// LS Electric XG5000 project: LoadWizardPro_v2
// PLC LoadWizardPLC
// module base 0 slot 0: FEnet:XGL-EFMT(B) (Fast Ethernet Module, Electrical Master)
// module base 0 slot 1: Input Module:XGI-D22A/B (DC 24V Input, 16 Contacts)
// module base 0 slot 2: Output Module:XGQ-TR2A/B (Transistor Output, 16 Contacts (0.5A, Sink Output/Source Output))
// module base 0 slot 3: Input Module:XGI-D22A/B (DC 24V Input, 16 Contacts)
// module base 0 slot 4: Output Module:XGQ-RY2A/B (Relay Output, 16 Contacts (2A, No Varistor/Varistor))

PROGRAM Main (task: Scan Program)

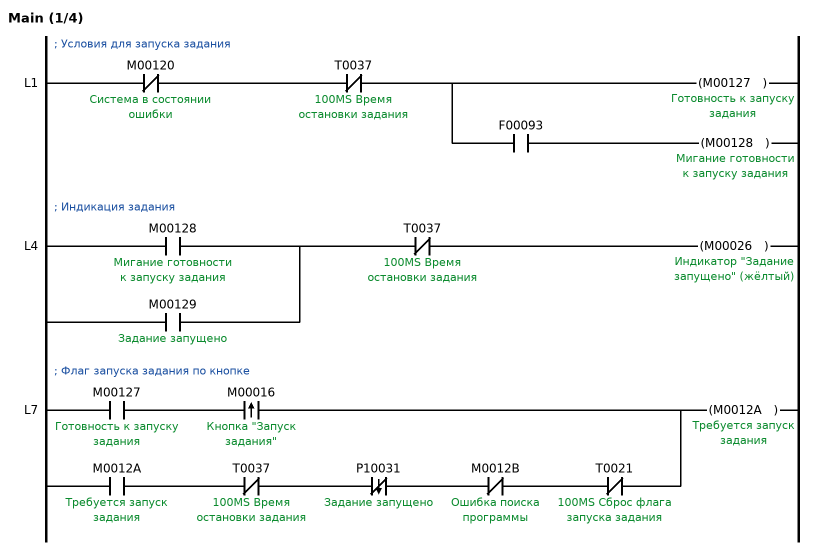
// Условия для запуска задания
; L1
LOAD NOT  M00120	// Система в состоянии ошибки
AND NOT   T0037	// 100MS Время остановки задания
OUT       M00127	// Готовность к запуску задания
AND       F00093
OUT       M00128	// Мигание готовности к запуску задания
// Индикация задания
; L4
LOAD      M00128	// Мигание готовности к запуску задания
OR        M00129	// Задание запущено
AND NOT   T0037	// 100MS Время остановки задания
OUT       M00026	// Индикатор "Задание запущено" (жёлтый)
// Флаг запуска задания по кнопке
; L7
LOAD      M00127	// Готовность к запуску задания
ANDP      M00016	// Кнопка "Запуск задания"
LOAD      M0012A	// Требуется запуск задания
AND NOT   T0037	// 100MS Время остановки задания
ANDN NOT  P10031	// Задание запущено
AND NOT   M0012B	// Ошибка поиска программы
AND NOT   T0021	// 100MS Сброс флага запуска задания
OR LOAD
OUT       M0012A	// Требуется запуск задания

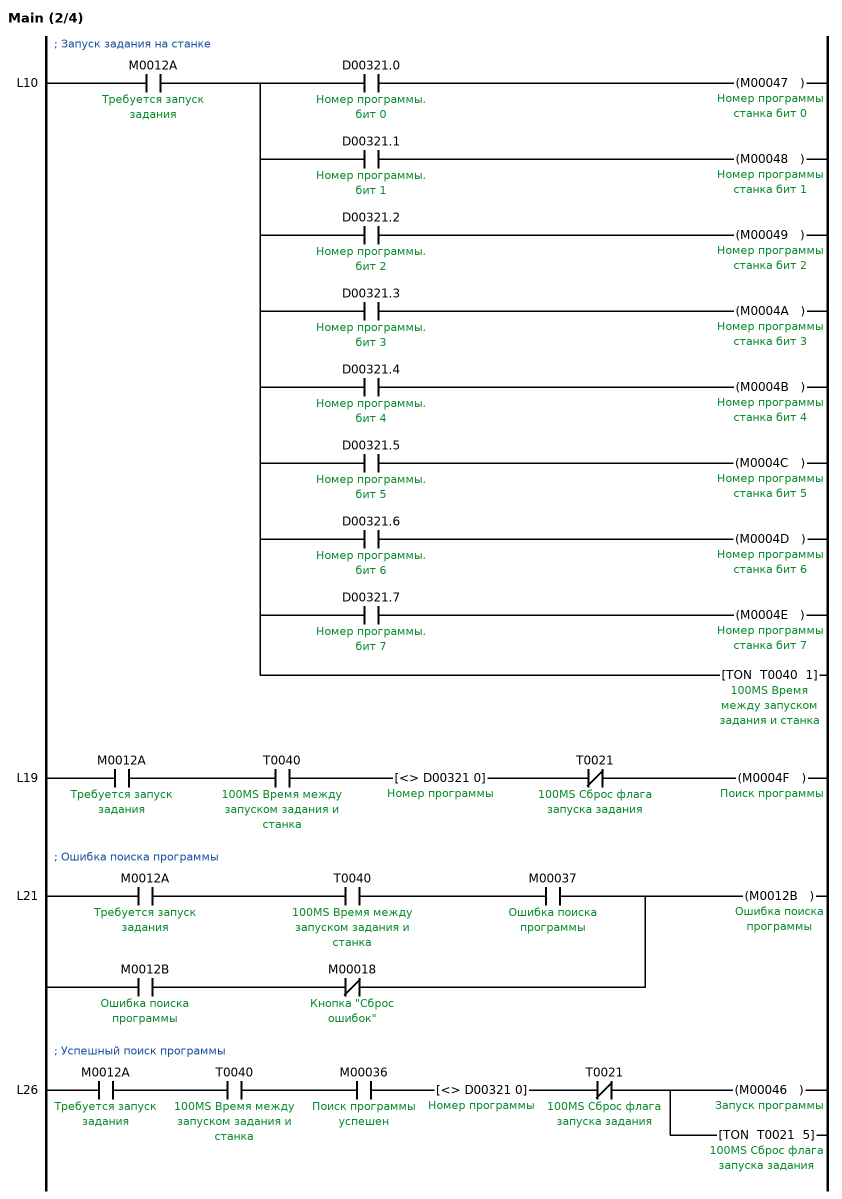
// Запуск задания на станке
; L10
LOAD      M0012A	// Требуется запуск задания
MPUSH
AND       D00321.0	// Номер программы. бит 0
OUT       M00047	// Номер программы станка бит 0
MLOAD
AND       D00321.1	// Номер программы. бит 1
OUT       M00048	// Номер программы станка бит 1
MLOAD
AND       D00321.2	// Номер программы. бит 2
OUT       M00049	// Номер программы станка бит 2
MLOAD
AND       D00321.3	// Номер программы. бит 3
OUT       M0004A	// Номер программы станка бит 3
MLOAD
AND       D00321.4	// Номер программы. бит 4
OUT       M0004B	// Номер программы станка бит 4
MLOAD
AND       D00321.5	// Номер программы. бит 5
OUT       M0004C	// Номер программы станка бит 5
MLOAD
AND       D00321.6	// Номер программы. бит 6
OUT       M0004D	// Номер программы станка бит 6
MLOAD
AND       D00321.7	// Номер программы. бит 7
OUT       M0004E	// Номер программы станка бит 7
MPOP
TON       T0040 1	// 100MS Время между запуском задания и станка
; L19
LOAD      M0012A	// Требуется запуск задания
AND       T0040	// 100MS Время между запуском задания и станка
AND<>     D00321 0	// Номер программы
AND NOT   T0021	// 100MS Сброс флага запуска задания
OUT       M0004F	// Поиск программы
// Ошибка поиска программы
; L21
LOAD      M0012A	// Требуется запуск задания
AND       T0040	// 100MS Время между запуском задания и станка
AND       M00037	// Ошибка поиска программы
LOAD      M0012B	// Ошибка поиска программы
AND NOT   M00018	// Кнопка "Сброс ошибок"
OR LOAD
OUT       M0012B	// Ошибка поиска программы
// Успешный поиск программы
; L26
LOAD      M0012A	// Требуется запуск задания
AND       T0040	// 100MS Время между запуском задания и станка
AND       M00036	// Поиск программы успешен
AND<>     D00321 0	// Номер программы
AND NOT   T0021	// 100MS Сброс флага запуска задания
OUT       M00046	// Запуск программы
TON       T0021 5	// 100MS Сброс флага запуска задания

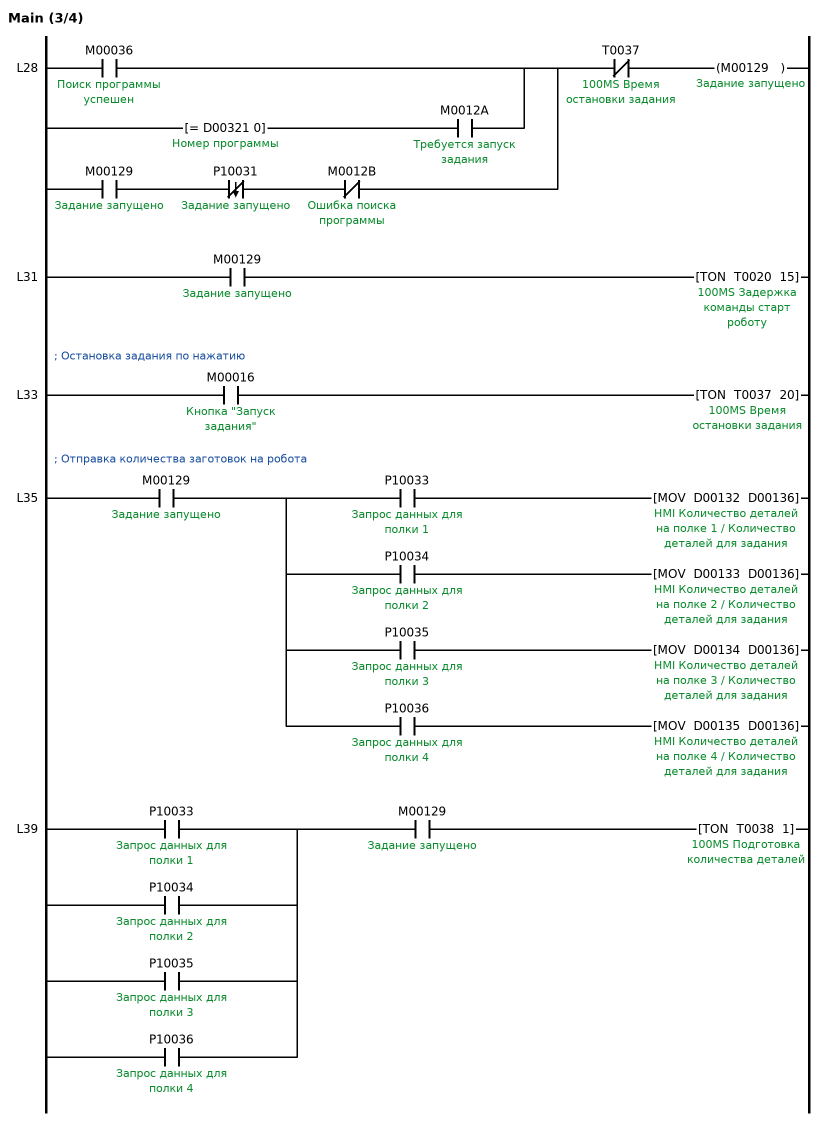
; L28
LOAD      M00036	// Поиск программы успешен
LOAD=     D00321 0	// Номер программы
AND       M0012A	// Требуется запуск задания
OR LOAD
LOAD      M00129	// Задание запущено
ANDN NOT  P10031	// Задание запущено
AND NOT   M0012B	// Ошибка поиска программы
OR LOAD
AND NOT   T0037	// 100MS Время остановки задания
OUT       M00129	// Задание запущено
; L31
LOAD      M00129	// Задание запущено
TON       T0020 15	// 100MS Задержка команды старт роботу
// Остановка задания по нажатию
; L33
LOAD      M00016	// Кнопка "Запуск задания"
TON       T0037 20	// 100MS Время остановки задания
// Отправка количества заготовок на робота
; L35
LOAD      M00129	// Задание запущено
MPUSH
AND       P10033	// Запрос данных для полки 1
MOV       D00132 D00136	// HMI Количество деталей на полке 1 / Количество деталей для задания
MLOAD
AND       P10034	// Запрос данных для полки 2
MOV       D00133 D00136	// HMI Количество деталей на полке 2 / Количество деталей для задания
MLOAD
AND       P10035	// Запрос данных для полки 3
MOV       D00134 D00136	// HMI Количество деталей на полке 3 / Количество деталей для задания
MPOP
AND       P10036	// Запрос данных для полки 4
MOV       D00135 D00136	// HMI Количество деталей на полке 4 / Количество деталей для задания
; L39
LOAD      P10033	// Запрос данных для полки 1
OR        P10034	// Запрос данных для полки 2
OR        P10035	// Запрос данных для полки 3
OR        P10036	// Запрос данных для полки 4
AND       M00129	// Задание запущено
TON       T0038 1	// 100MS Подготовка количества деталей

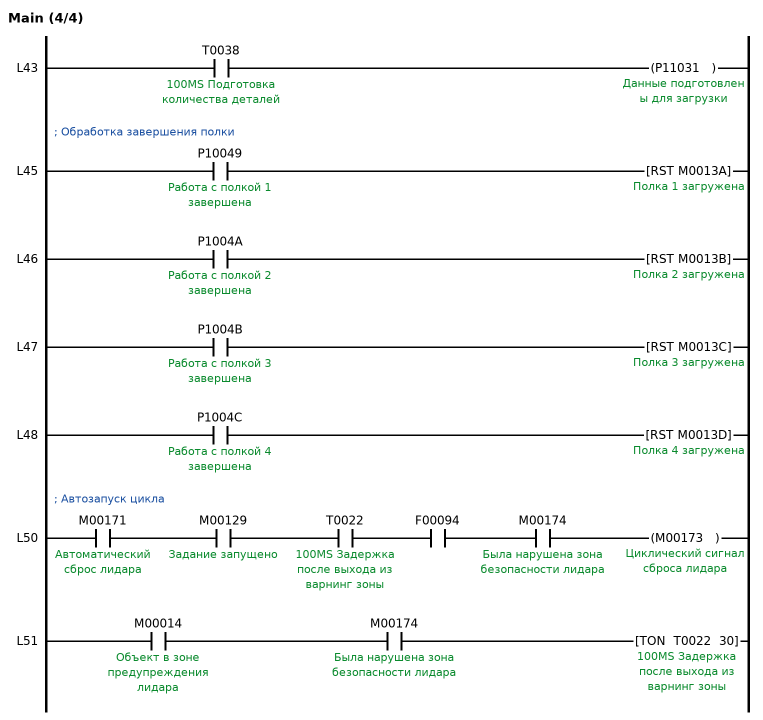
; L43
LOAD      T0038	// 100MS Подготовка количества деталей
OUT       P11031	// Данные подготовлены для загрузки
// Обработка завершения полки
; L45
LOAD      P10049	// Работа с полкой 1 завершена
RST       M0013A	// Полка 1 загружена
; L46
LOAD      P1004A	// Работа с полкой 2 завершена
RST       M0013B	// Полка 2 загружена
; L47
LOAD      P1004B	// Работа с полкой 3 завершена
RST       M0013C	// Полка 3 загружена
; L48
LOAD      P1004C	// Работа с полкой 4 завершена
RST       M0013D	// Полка 4 загружена
// Автозапуск цикла
; L50
LOAD      M00171	// Автоматический сброс лидара
AND       M00129	// Задание запущено
AND       T0022	// 100MS Задержка после выхода из варнинг зоны
AND       F00094
AND       M00174	// Была нарушена зона безопасности лидара
OUT       M00173	// Циклический сигнал сброса лидара
; L51
LOAD      M00014	// Объект в зоне предупреждения лидара
AND       M00174	// Была нарушена зона безопасности лидара
TON       T0022 30	// 100MS Задержка после выхода из варнинг зоны

PROGRAM Robot (task: Scan Program)

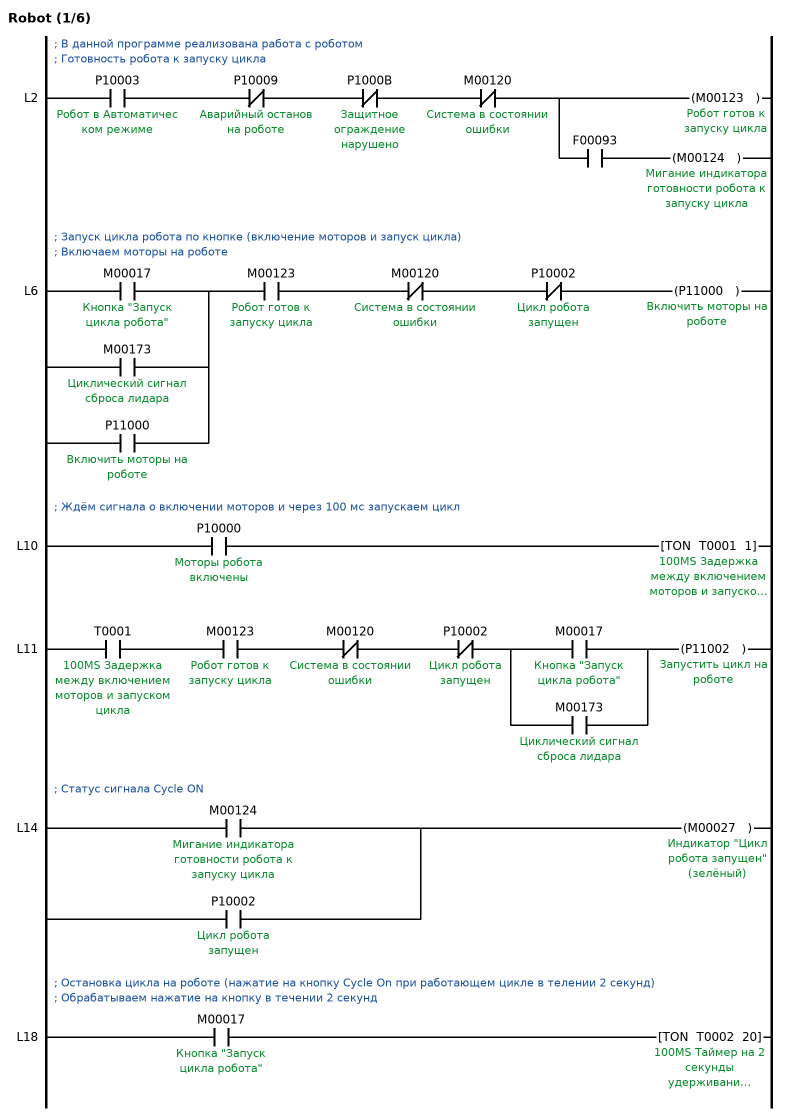
// В данной программе реализована работа с роботом
// Готовность робота к запуску цикла
; L2
LOAD      P10003	// Робот в Автоматическом режиме
AND NOT   P10009	// Аварийный останов на роботе
AND NOT   P1000B	// Защитное ограждение нарушено
AND NOT   M00120	// Система в состоянии ошибки
OUT       M00123	// Робот готов к запуску цикла
AND       F00093
OUT       M00124	// Мигание индикатора готовности робота к запуску цикла
// Запуск цикла робота по кнопке (включение моторов и запуск цикла)
// Включаем моторы на роботе
; L6
LOAD      M00017	// Кнопка "Запуск цикла робота"
OR        M00173	// Циклический сигнал сброса лидара
OR        P11000	// Включить моторы на роботе
AND       M00123	// Робот готов к запуску цикла
AND NOT   M00120	// Система в состоянии ошибки
AND NOT   P10002	// Цикл робота запущен
OUT       P11000	// Включить моторы на роботе
// Ждём сигнала о включении моторов и через 100 мс запускаем цикл
; L10
LOAD      P10000	// Моторы робота включены
TON       T0001 1	// 100MS Задержка между включением моторов и запуском цикла
; L11
LOAD      T0001	// 100MS Задержка между включением моторов и запуском цикла
AND       M00123	// Робот готов к запуску цикла
AND NOT   M00120	// Система в состоянии ошибки
AND NOT   P10002	// Цикл робота запущен
LOAD      M00017	// Кнопка "Запуск цикла робота"
OR        M00173	// Циклический сигнал сброса лидара
AND LOAD
OUT       P11002	// Запустить цикл на роботе
// output comment: 
// Статус сигнала Cycle ON
; L14
LOAD      M00124	// Мигание индикатора готовности робота к запуску цикла
OR        P10002	// Цикл робота запущен
OUT       M00027	// Индикатор "Цикл робота запущен" (зелёный)
// Остановка цикла на роботе (нажатие на кнопку Cycle On при работающем цикле в телении 2 секунд)
// Обрабатываем нажатие на кнопку в течении 2 секунд
; L18
LOAD      M00017	// Кнопка "Запуск цикла робота"
TON       T0002 20	// 100MS Таймер на 2 секунды удерживания кнопки

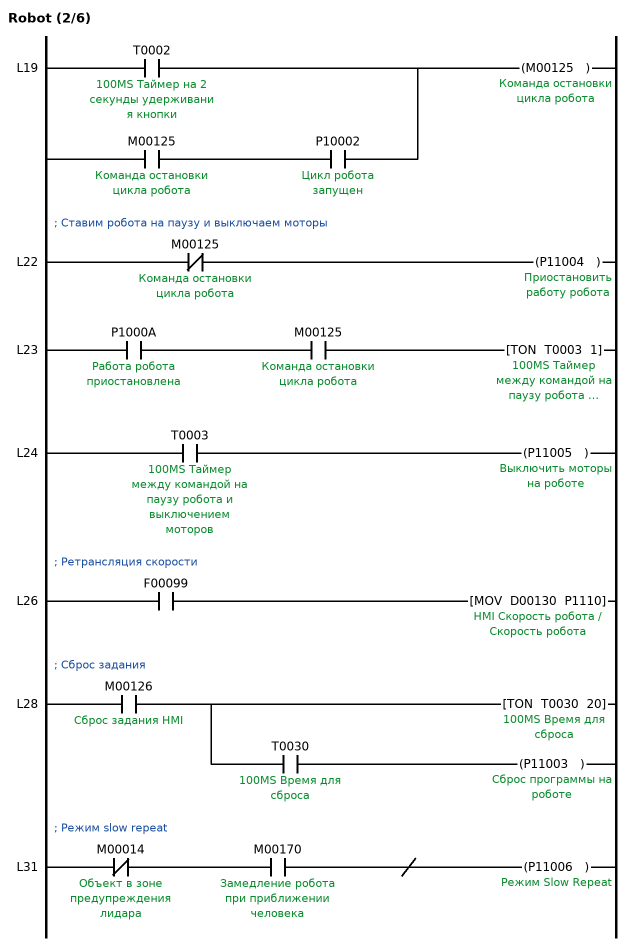
; L19
LOAD      T0002	// 100MS Таймер на 2 секунды удерживания кнопки
LOAD      M00125	// Команда остановки цикла робота
AND       P10002	// Цикл робота запущен
OR LOAD
OUT       M00125	// Команда остановки цикла робота
// Ставим робота на паузу и выключаем моторы
; L22
LOAD NOT  M00125	// Команда остановки цикла робота
OUT       P11004	// Приостановить работу робота
; L23
LOAD      P1000A	// Работа робота приостановлена
AND       M00125	// Команда остановки цикла робота
TON       T0003 1	// 100MS Таймер между командой на паузу робота и выключением моторов
; L24
LOAD      T0003	// 100MS Таймер между командой на паузу робота и выключением моторов
OUT       P11005	// Выключить моторы на роботе
// Ретрансляция скорости
; L26
LOAD      F00099
MOV       D00130 P1110	// HMI Скорость робота / Скорость робота
// Сброс задания
; L28
LOAD      M00126	// Сброс задания HMI
TON       T0030 20	// 100MS Время для сброса
AND       T0030	// 100MS Время для сброса
OUT       P11003	// Сброс программы на роботе
// Режим slow repeat
; L31
LOAD NOT  M00014	// Объект в зоне предупреждения лидара
AND       M00170	// Замедление робота при приближении человека
NOT
OUT       P11006	// Режим Slow Repeat

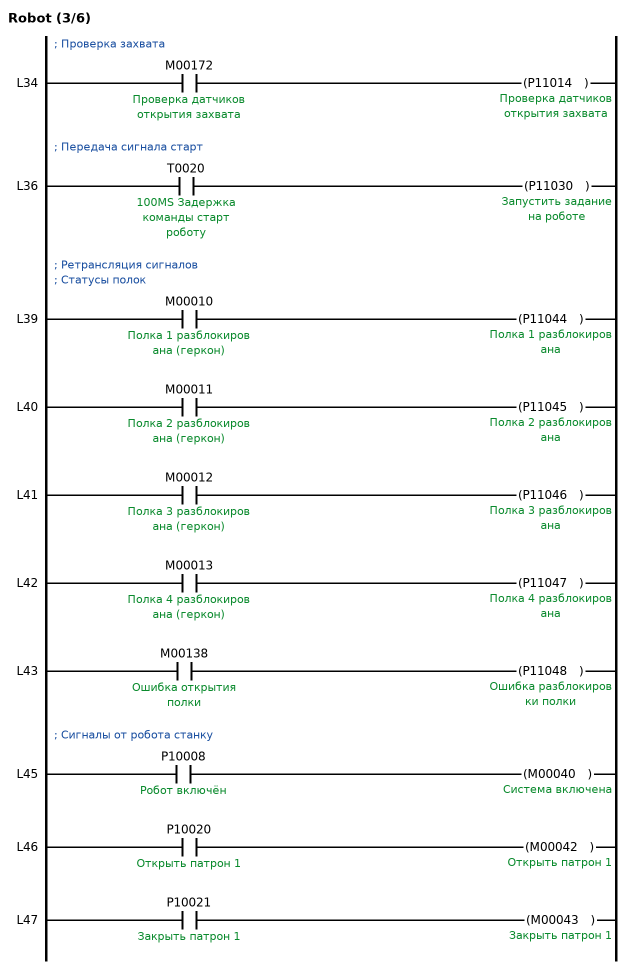
// Проверка захвата
; L34
LOAD      M00172	// Проверка датчиков открытия захвата
OUT       P11014	// Проверка датчиков открытия захвата
// Передача сигнала старт
; L36
LOAD      T0020	// 100MS Задержка команды старт роботу
OUT       P11030	// Запустить задание на роботе
// Ретрансляция сигналов
// Статусы полок
; L39
LOAD      M00010	// Полка 1 разблокирована (геркон)
OUT       P11044	// Полка 1 разблокирована
; L40
LOAD      M00011	// Полка 2 разблокирована (геркон)
OUT       P11045	// Полка 2 разблокирована
; L41
LOAD      M00012	// Полка 3 разблокирована (геркон)
OUT       P11046	// Полка 3 разблокирована
; L42
LOAD      M00013	// Полка 4 разблокирована (геркон)
OUT       P11047	// Полка 4 разблокирована
; L43
LOAD      M00138	// Ошибка открытия полки
OUT       P11048	// Ошибка разблокировки полки
// Сигналы от робота станку
; L45
LOAD      P10008	// Робот включён
OUT       M00040	// Система включена
; L46
LOAD      P10020	// Открыть патрон 1
OUT       M00042	// Открыть патрон 1
; L47
LOAD      P10021	// Закрыть патрон 1
OUT       M00043	// Закрыть патрон 1

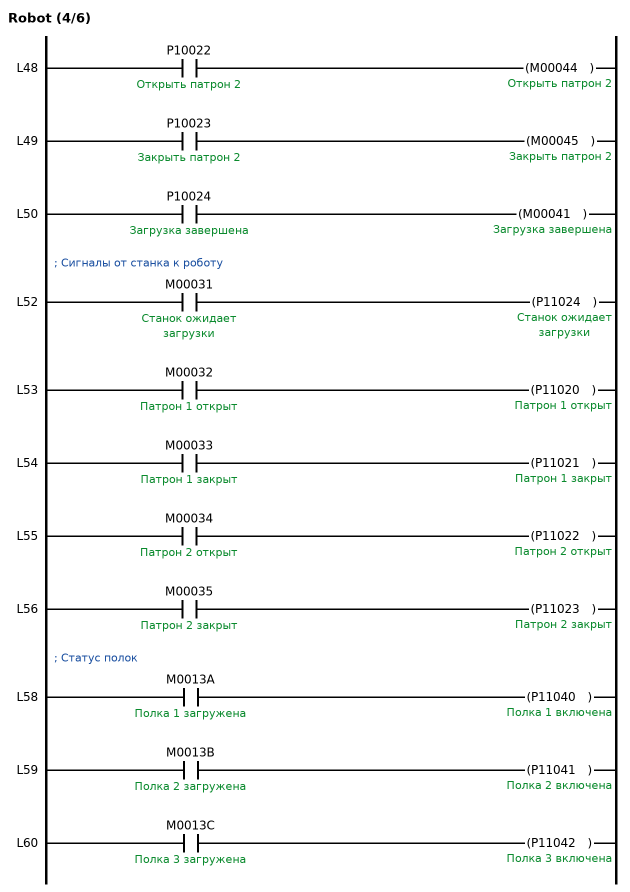
; L48
LOAD      P10022	// Открыть патрон 2
OUT       M00044	// Открыть патрон 2
; L49
LOAD      P10023	// Закрыть патрон 2
OUT       M00045	// Закрыть патрон 2
; L50
LOAD      P10024	// Загрузка завершена
OUT       M00041	// Загрузка завершена
// Сигналы от станка к роботу
; L52
LOAD      M00031	// Станок ожидает загрузки
OUT       P11024	// Станок ожидает загрузки
; L53
LOAD      M00032	// Патрон 1 открыт
OUT       P11020	// Патрон 1 открыт
; L54
LOAD      M00033	// Патрон 1 закрыт
OUT       P11021	// Патрон 1 закрыт
; L55
LOAD      M00034	// Патрон 2 открыт
OUT       P11022	// Патрон 2 открыт
; L56
LOAD      M00035	// Патрон 2 закрыт
OUT       P11023	// Патрон 2 закрыт
// Статус полок
; L58
LOAD      M0013A	// Полка 1 загружена
OUT       P11040	// Полка 1 включена
; L59
LOAD      M0013B	// Полка 2 загружена
OUT       P11041	// Полка 2 включена
; L60
LOAD      M0013C	// Полка 3 загружена
OUT       P11042	// Полка 3 включена

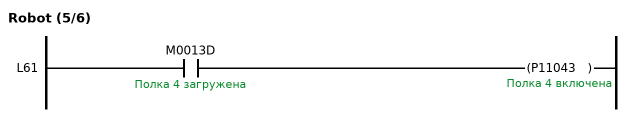
; L61
LOAD      M0013D	// Полка 4 загружена
OUT       P11043	// Полка 4 включена

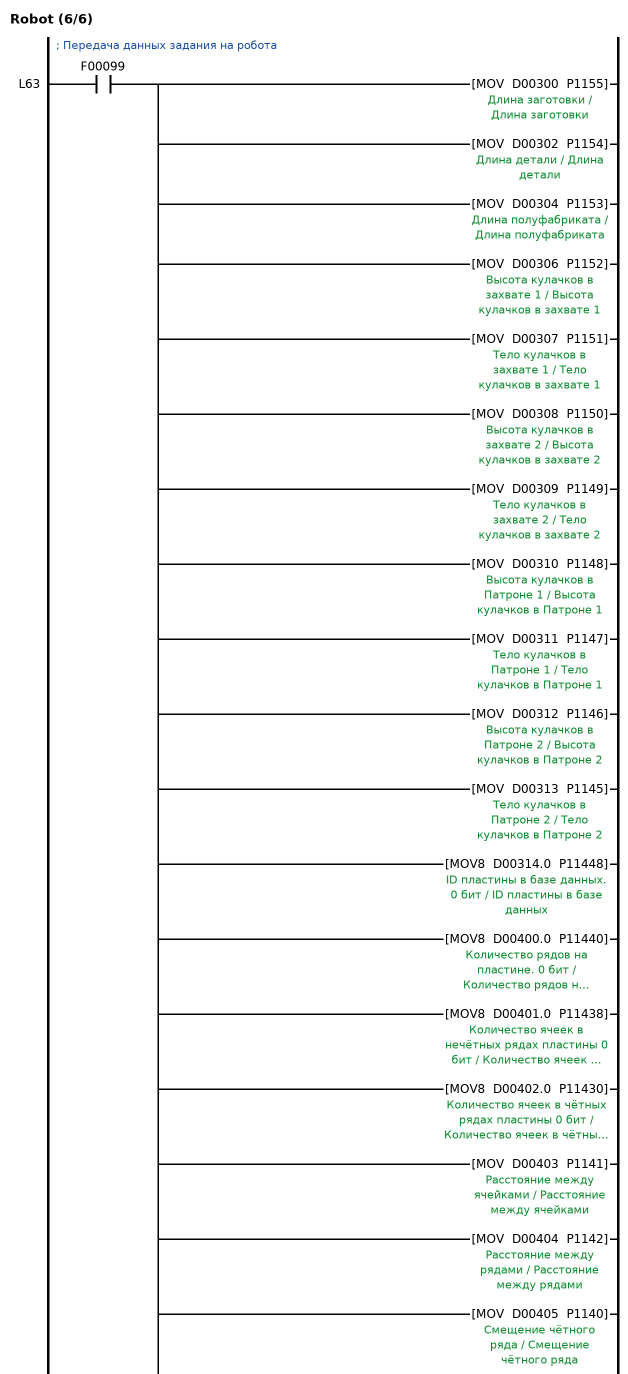

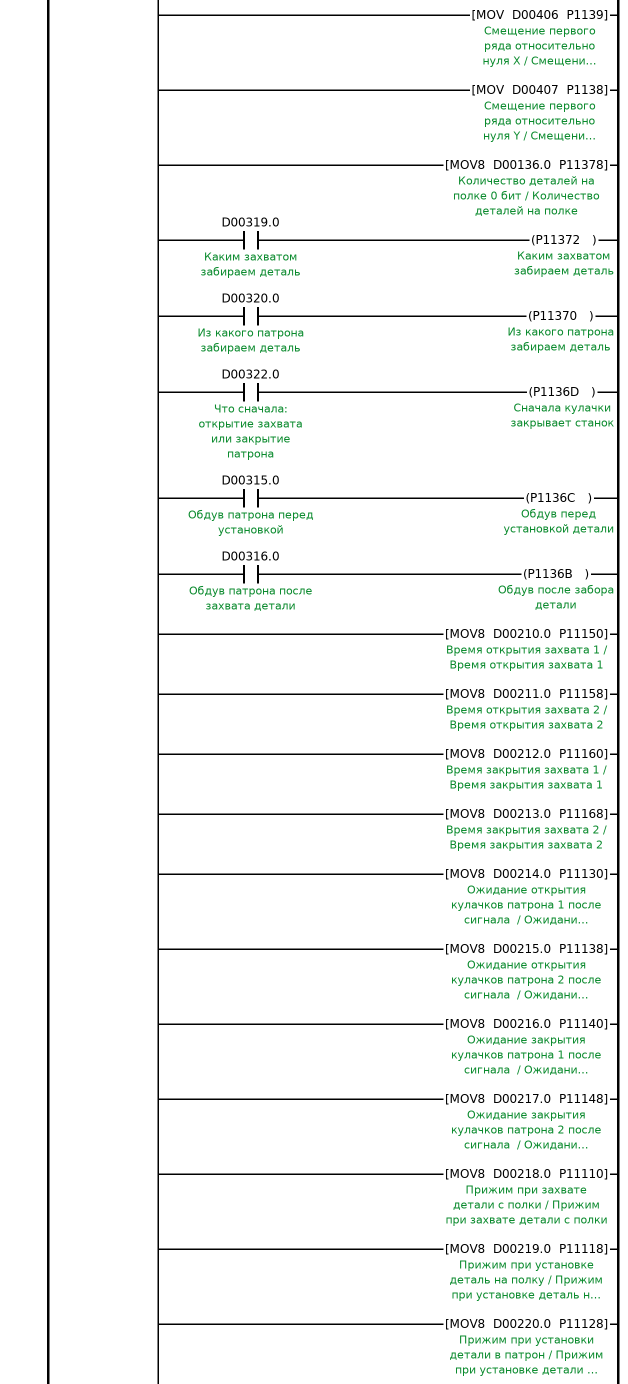

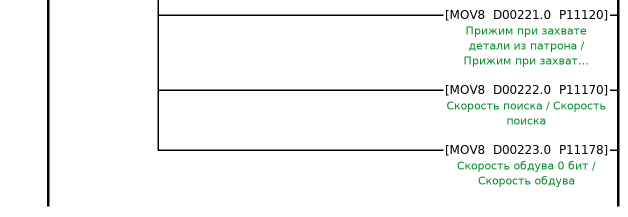
// Передача данных задания на робота
; L63
LOAD      F00099
MOV       D00300 P1155	// Длина заготовки / Длина заготовки
MOV       D00302 P1154	// Длина детали / Длина детали
MOV       D00304 P1153	// Длина полуфабриката / Длина полуфабриката
MOV       D00306 P1152	// Высота кулачков в захвате 1 / Высота кулачков в захвате 1
MOV       D00307 P1151	// Тело кулачков в захвате 1 / Тело кулачков в захвате 1
MOV       D00308 P1150	// Высота кулачков в захвате 2 / Высота кулачков в захвате 2
MOV       D00309 P1149	// Тело кулачков в захвате 2 / Тело кулачков в захвате 2
MOV       D00310 P1148	// Высота кулачков в Патроне 1 / Высота кулачков в Патроне 1
MOV       D00311 P1147	// Тело кулачков в Патроне 1 / Тело кулачков в Патроне 1
MOV       D00312 P1146	// Высота кулачков в Патроне 2 / Высота кулачков в Патроне 2
MOV       D00313 P1145	// Тело кулачков в Патроне 2 / Тело кулачков в Патроне 2
MOV8      D00314.0 P11448	// ID пластины в базе данных. 0 бит / ID пластины в базе данных
MOV8      D00400.0 P11440	// Количество рядов на пластине. 0 бит / Количество рядов на пластине
MOV8      D00401.0 P11438	// Количество ячеек в нечётных рядах пластины 0 бит / Количество ячеек в нечётных рядах пластины
MOV8      D00402.0 P11430	// Количество ячеек в чётных рядах пластины 0 бит / Количество ячеек в чётных рядах пластины
MOV       D00403 P1141	// Расстояние между ячейками / Расстояние между ячейками
MOV       D00404 P1142	// Расстояние между рядами / Расстояние между рядами
MOV       D00405 P1140	// Смещение чётного ряда / Смещение чётного ряда
MOV       D00406 P1139	// Смещение первого ряда относительно нуля Х / Смещение первого ряда относительно нуля Х
MOV       D00407 P1138	// Смещение первого ряда относительно нуля Y / Смещение первого ряда относительно нуля Y
MOV8      D00136.0 P11378	// Количество деталей на полке 0 бит / Количество деталей на полке
MPUSH
AND       D00319.0	// Каким захватом забираем деталь
OUT       P11372	// Каким захватом забираем деталь
MLOAD
AND       D00320.0	// Из какого патрона забираем деталь
OUT       P11370	// Из какого патрона забираем деталь
MLOAD
AND       D00322.0	// Что сначала: открытие захвата или закрытие патрона  
OUT       P1136D	// Сначала кулачки закрывает станок
MLOAD
AND       D00315.0	// Обдув патрона перед установкой
OUT       P1136C	// Обдув перед установкой детали
MLOAD
AND       D00316.0	// Обдув патрона после захвата детали
OUT       P1136B	// Обдув после забора детали
MPOP
MOV8      D00210.0 P11150	// Время открытия захвата 1 / Время открытия захвата 1
MOV8      D00211.0 P11158	// Время открытия захвата 2 / Время открытия захвата 2
MOV8      D00212.0 P11160	// Время закрытия захвата 1 / Время закрытия захвата 1
MOV8      D00213.0 P11168	// Время закрытия захвата 2 / Время закрытия захвата 2
MOV8      D00214.0 P11130	// Ожидание открытия кулачков патрона 1 после сигнала  / Ожидание открытия кулачков патрона 1 после сигнала 
MOV8      D00215.0 P11138	// Ожидание открытия кулачков патрона 2 после сигнала  / Ожидание открытия кулачков патрона 2 после сигнала 
MOV8      D00216.0 P11140	// Ожидание закрытия кулачков патрона 1 после сигнала  / Ожидание закрытия кулачков патрона 1 после сигнала 
MOV8      D00217.0 P11148	// Ожидание закрытия кулачков патрона 2 после сигнала  / Ожидание закрытия кулачков патрона 2 после сигнала 
MOV8      D00218.0 P11110	// Прижим при захвате детали с полки / Прижим при захвате детали с полки
MOV8      D00219.0 P11118	// Прижим при установке деталь на полку / Прижим при установке деталь на полку
MOV8      D00220.0 P11128	// Прижим при установки детали в патрон / Прижим при установке детали в патрон
MOV8      D00221.0 P11120	// Прижим при захвате детали из патрона / Прижим при захвате детали из патрона
MOV8      D00222.0 P11170	// Скорость поиска / Скорость поиска
MOV8      D00223.0 P11178	// Скорость обдува 0 бит / Скорость обдува

PROGRAM IO (task: Scan Program)

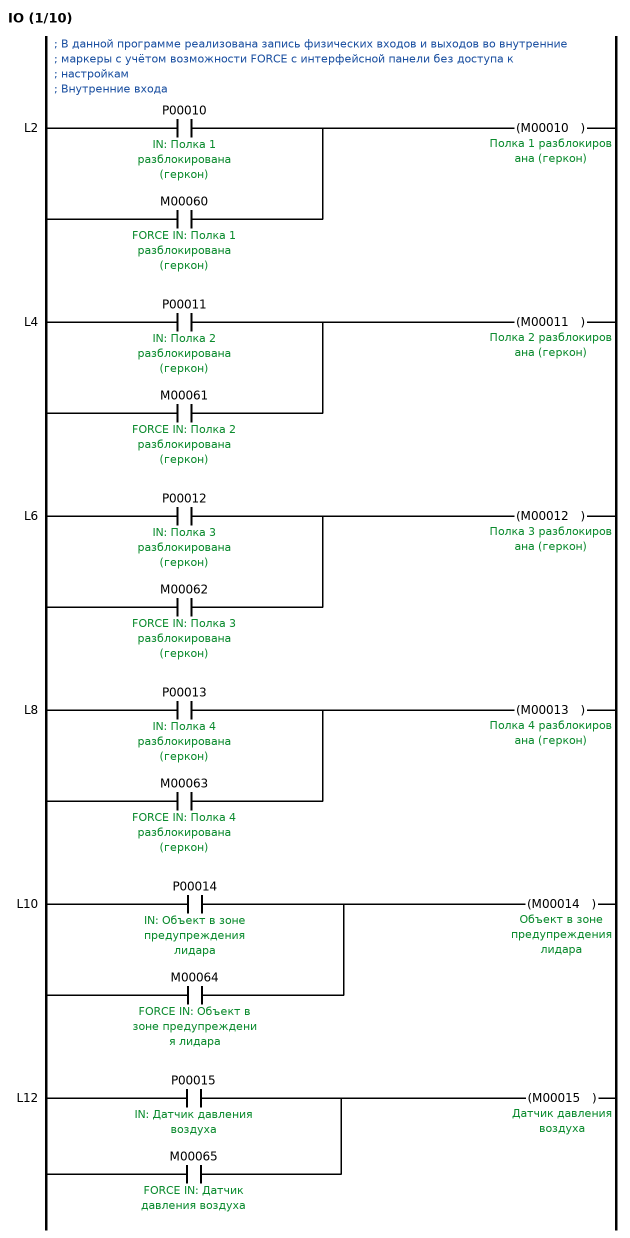
// В данной программе реализована запись физических входов и выходов во внутренние маркеры с учётом возможности FORCE с интерфейсной панели без доступа к настройкам
// Внутренние входа
; L2
LOAD      P00010	// IN: Полка 1 разблокирована (геркон)
OR        M00060	// FORCE IN: Полка 1 разблокирована (геркон)
OUT       M00010	// Полка 1 разблокирована (геркон)
; L4
LOAD      P00011	// IN: Полка 2 разблокирована (геркон)
OR        M00061	// FORCE IN: Полка 2 разблокирована (геркон)
OUT       M00011	// Полка 2 разблокирована (геркон)
; L6
LOAD      P00012	// IN: Полка 3 разблокирована (геркон)
OR        M00062	// FORCE IN: Полка 3 разблокирована (геркон)
OUT       M00012	// Полка 3 разблокирована (геркон)
; L8
LOAD      P00013	// IN: Полка 4 разблокирована (геркон)
OR        M00063	// FORCE IN: Полка 4 разблокирована (геркон)
OUT       M00013	// Полка 4 разблокирована (геркон)
; L10
LOAD      P00014	// IN: Объект в зоне предупреждения лидара
OR        M00064	// FORCE IN: Объект в зоне предупреждения лидара
OUT       M00014	// Объект в зоне предупреждения лидара
; L12
LOAD      P00015	// IN: Датчик давления воздуха
OR        M00065	// FORCE IN: Датчик давления воздуха
OUT       M00015	// Датчик давления воздуха

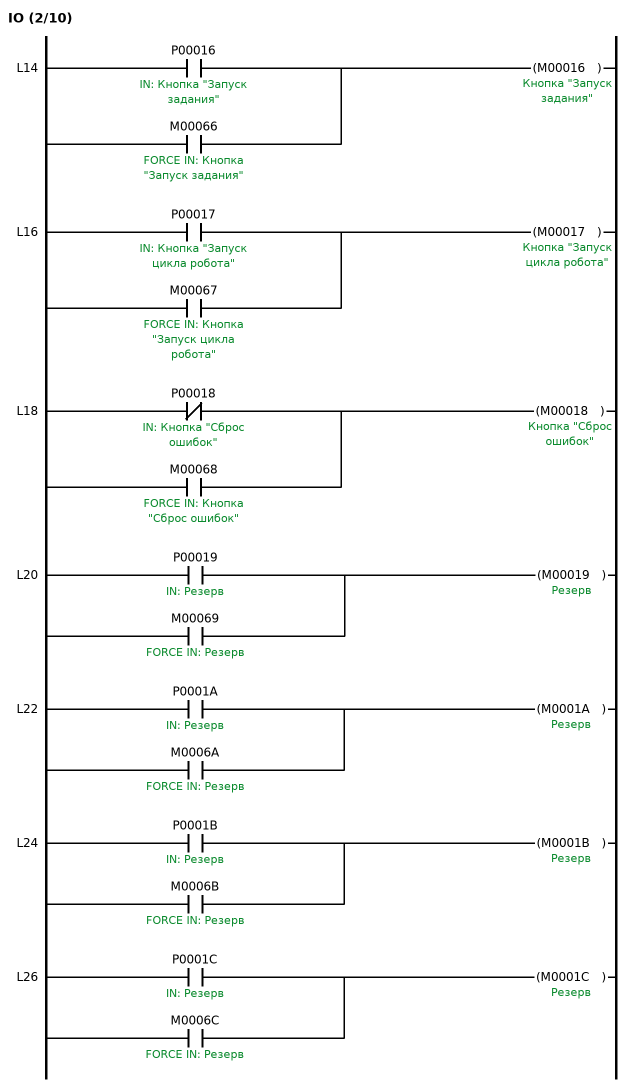
; L14
LOAD      P00016	// IN: Кнопка "Запуск задания"
OR        M00066	// FORCE IN: Кнопка "Запуск задания"
OUT       M00016	// Кнопка "Запуск задания"
; L16
LOAD      P00017	// IN: Кнопка "Запуск цикла робота"
OR        M00067	// FORCE IN: Кнопка "Запуск цикла робота"
OUT       M00017	// Кнопка "Запуск цикла робота"
; L18
LOAD NOT  P00018	// IN: Кнопка "Сброс ошибок"
OR        M00068	// FORCE IN: Кнопка "Сброс ошибок"
OUT       M00018	// Кнопка "Сброс ошибок"
; L20
LOAD      P00019	// IN: Резерв
OR        M00069	// FORCE IN: Резерв
OUT       M00019	// Резерв
; L22
LOAD      P0001A	// IN: Резерв
OR        M0006A	// FORCE IN: Резерв
OUT       M0001A	// Резерв
; L24
LOAD      P0001B	// IN: Резерв
OR        M0006B	// FORCE IN: Резерв
OUT       M0001B	// Резерв
; L26
LOAD      P0001C	// IN: Резерв
OR        M0006C	// FORCE IN: Резерв
OUT       M0001C	// Резерв

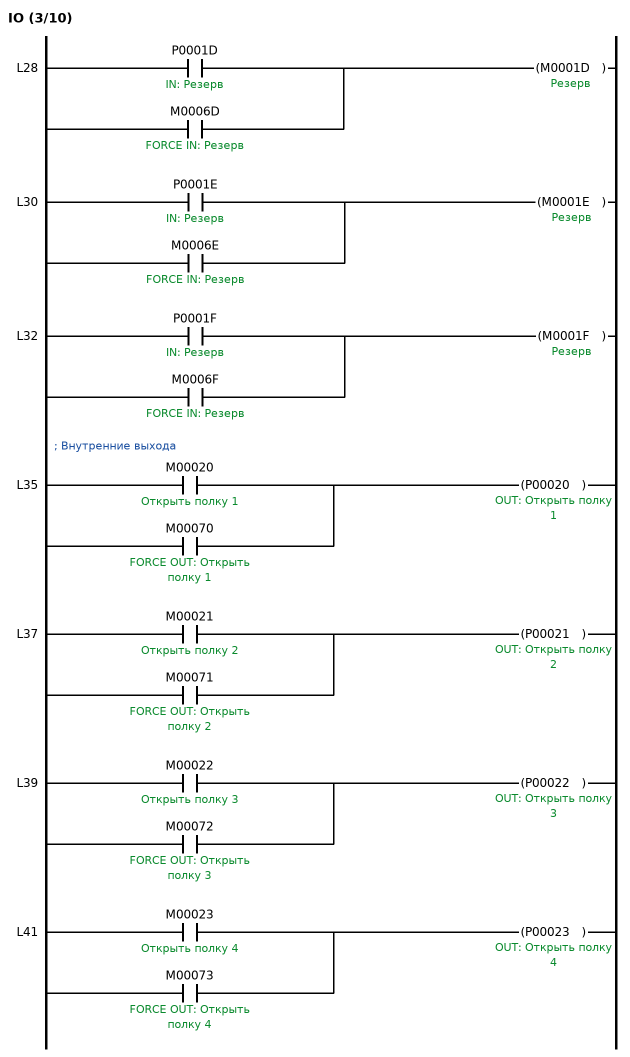
; L28
LOAD      P0001D	// IN: Резерв
OR        M0006D	// FORCE IN: Резерв
OUT       M0001D	// Резерв
; L30
LOAD      P0001E	// IN: Резерв
OR        M0006E	// FORCE IN: Резерв
OUT       M0001E	// Резерв
; L32
LOAD      P0001F	// IN: Резерв
OR        M0006F	// FORCE IN: Резерв
OUT       M0001F	// Резерв
// Внутренние выхода
; L35
LOAD      M00020	// Открыть полку 1
OR        M00070	// FORCE OUT: Открыть полку 1
OUT       P00020	// OUT: Открыть полку 1
; L37
LOAD      M00021	// Открыть полку 2
OR        M00071	// FORCE OUT: Открыть полку 2
OUT       P00021	// OUT: Открыть полку 2
; L39
LOAD      M00022	// Открыть полку 3
OR        M00072	// FORCE OUT: Открыть полку 3
OUT       P00022	// OUT: Открыть полку 3
; L41
LOAD      M00023	// Открыть полку 4
OR        M00073	// FORCE OUT: Открыть полку 4
OUT       P00023	// OUT: Открыть полку 4

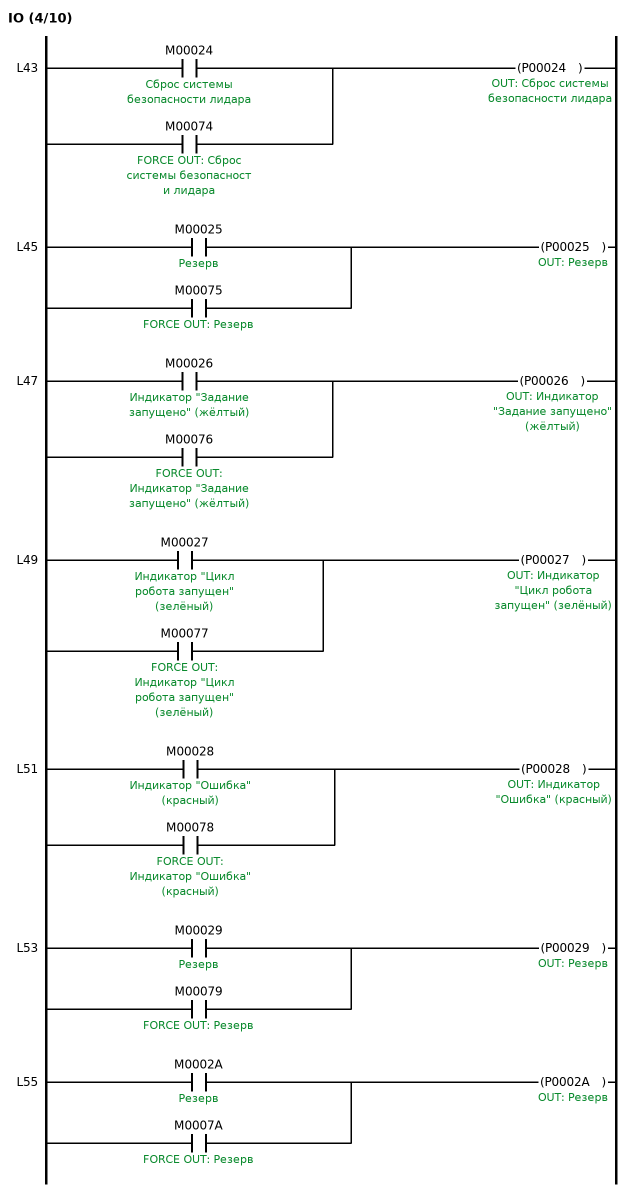
; L43
LOAD      M00024	// Сброс системы безопасности лидара
OR        M00074	// FORCE OUT: Сброс системы безопасности лидара
OUT       P00024	// OUT: Сброс системы безопасности лидара
; L45
LOAD      M00025	// Резерв
OR        M00075	// FORCE OUT: Резерв
OUT       P00025	// OUT: Резерв
; L47
LOAD      M00026	// Индикатор "Задание запущено" (жёлтый)
OR        M00076	// FORCE OUT: Индикатор "Задание запущено" (жёлтый)
OUT       P00026	// OUT: Индикатор "Задание запущено" (жёлтый)
; L49
LOAD      M00027	// Индикатор "Цикл робота запущен" (зелёный)
OR        M00077	// FORCE OUT: Индикатор "Цикл робота запущен" (зелёный)
OUT       P00027	// OUT: Индикатор "Цикл робота запущен" (зелёный)
; L51
LOAD      M00028	// Индикатор "Ошибка" (красный)
OR        M00078	// FORCE OUT: Индикатор "Ошибка" (красный)
OUT       P00028	// OUT: Индикатор "Ошибка" (красный)
; L53
LOAD      M00029	// Резерв
OR        M00079	// FORCE OUT: Резерв
OUT       P00029	// OUT: Резерв
; L55
LOAD      M0002A	// Резерв
OR        M0007A	// FORCE OUT: Резерв
OUT       P0002A	// OUT: Резерв

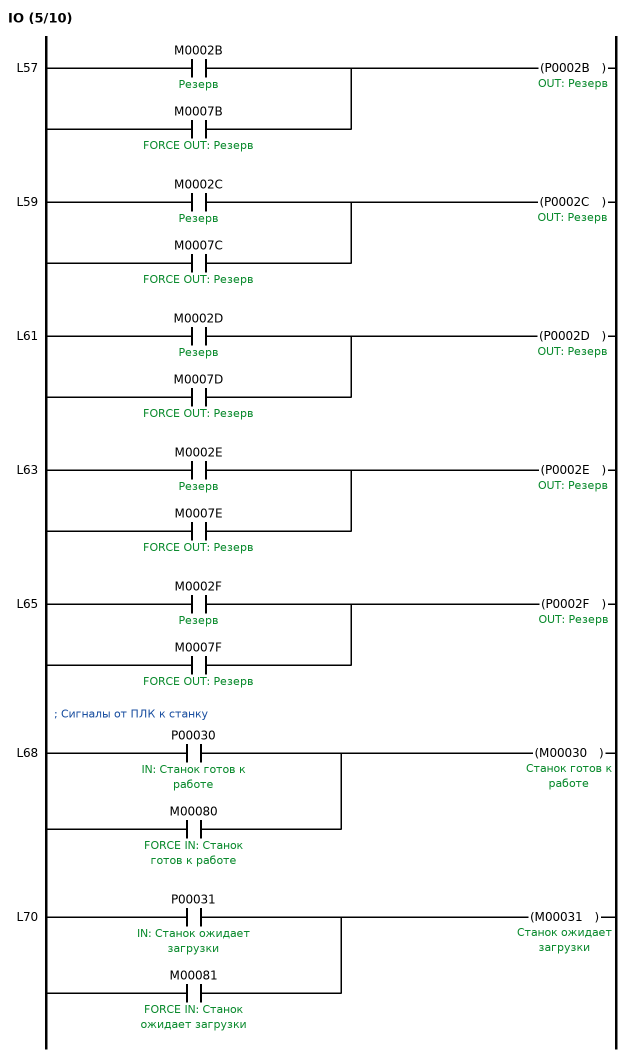
; L57
LOAD      M0002B	// Резерв
OR        M0007B	// FORCE OUT: Резерв
OUT       P0002B	// OUT: Резерв
; L59
LOAD      M0002C	// Резерв
OR        M0007C	// FORCE OUT: Резерв
OUT       P0002C	// OUT: Резерв
; L61
LOAD      M0002D	// Резерв
OR        M0007D	// FORCE OUT: Резерв
OUT       P0002D	// OUT: Резерв
; L63
LOAD      M0002E	// Резерв
OR        M0007E	// FORCE OUT: Резерв
OUT       P0002E	// OUT: Резерв
; L65
LOAD      M0002F	// Резерв
OR        M0007F	// FORCE OUT: Резерв
OUT       P0002F	// OUT: Резерв
// Сигналы от ПЛК к станку
; L68
LOAD      P00030	// IN: Станок готов к работе
OR        M00080	// FORCE IN: Станок готов к работе
OUT       M00030	// Станок готов к работе
; L70
LOAD      P00031	// IN: Станок ожидает загрузки
OR        M00081	// FORCE IN: Станок ожидает загрузки
OUT       M00031	// Станок ожидает загрузки

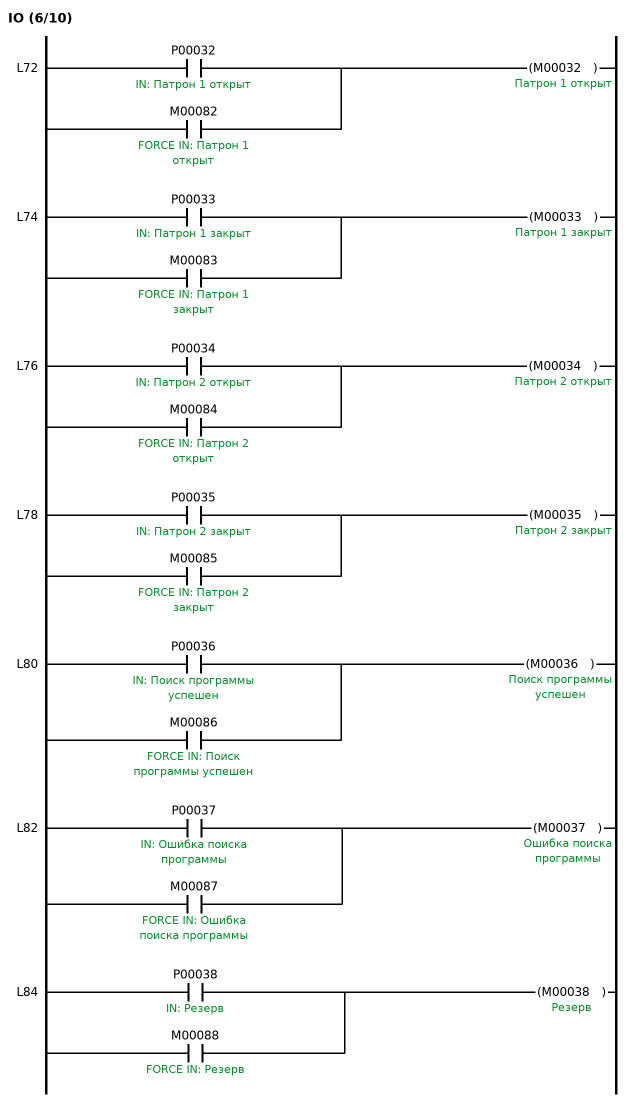
; L72
LOAD      P00032	// IN: Патрон 1 открыт
OR        M00082	// FORCE IN: Патрон 1 открыт
OUT       M00032	// Патрон 1 открыт
; L74
LOAD      P00033	// IN: Патрон 1 закрыт
OR        M00083	// FORCE IN: Патрон 1 закрыт
OUT       M00033	// Патрон 1 закрыт
; L76
LOAD      P00034	// IN: Патрон 2 открыт
OR        M00084	// FORCE IN: Патрон 2 открыт
OUT       M00034	// Патрон 2 открыт
; L78
LOAD      P00035	// IN: Патрон 2 закрыт
OR        M00085	// FORCE IN: Патрон 2 закрыт
OUT       M00035	// Патрон 2 закрыт
; L80
LOAD      P00036	// IN: Поиск программы успешен
OR        M00086	// FORCE IN: Поиск программы успешен
OUT       M00036	// Поиск программы успешен
; L82
LOAD      P00037	// IN: Ошибка поиска программы
OR        M00087	// FORCE IN: Ошибка поиска программы
OUT       M00037	// Ошибка поиска программы
; L84
LOAD      P00038	// IN: Резерв
OR        M00088	// FORCE IN: Резерв
OUT       M00038	// Резерв

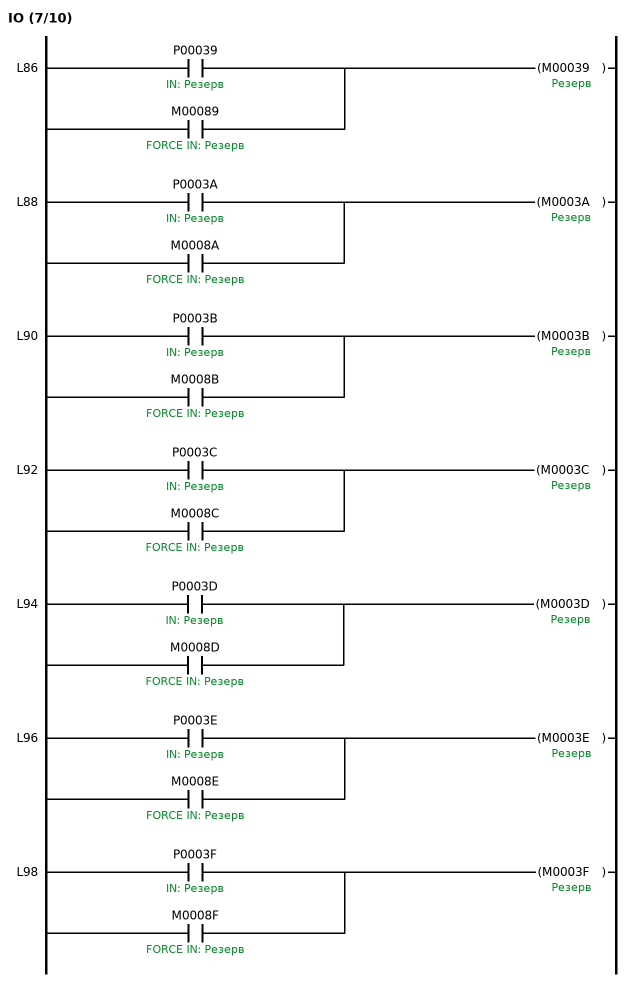
; L86
LOAD      P00039	// IN: Резерв
OR        M00089	// FORCE IN: Резерв
OUT       M00039	// Резерв
; L88
LOAD      P0003A	// IN: Резерв
OR        M0008A	// FORCE IN: Резерв
OUT       M0003A	// Резерв
; L90
LOAD      P0003B	// IN: Резерв
OR        M0008B	// FORCE IN: Резерв
OUT       M0003B	// Резерв
; L92
LOAD      P0003C	// IN: Резерв
OR        M0008C	// FORCE IN: Резерв
OUT       M0003C	// Резерв
; L94
LOAD      P0003D	// IN: Резерв
OR        M0008D	// FORCE IN: Резерв
OUT       M0003D	// Резерв
; L96
LOAD      P0003E	// IN: Резерв
OR        M0008E	// FORCE IN: Резерв
OUT       M0003E	// Резерв
; L98
LOAD      P0003F	// IN: Резерв
OR        M0008F	// FORCE IN: Резерв
OUT       M0003F	// Резерв

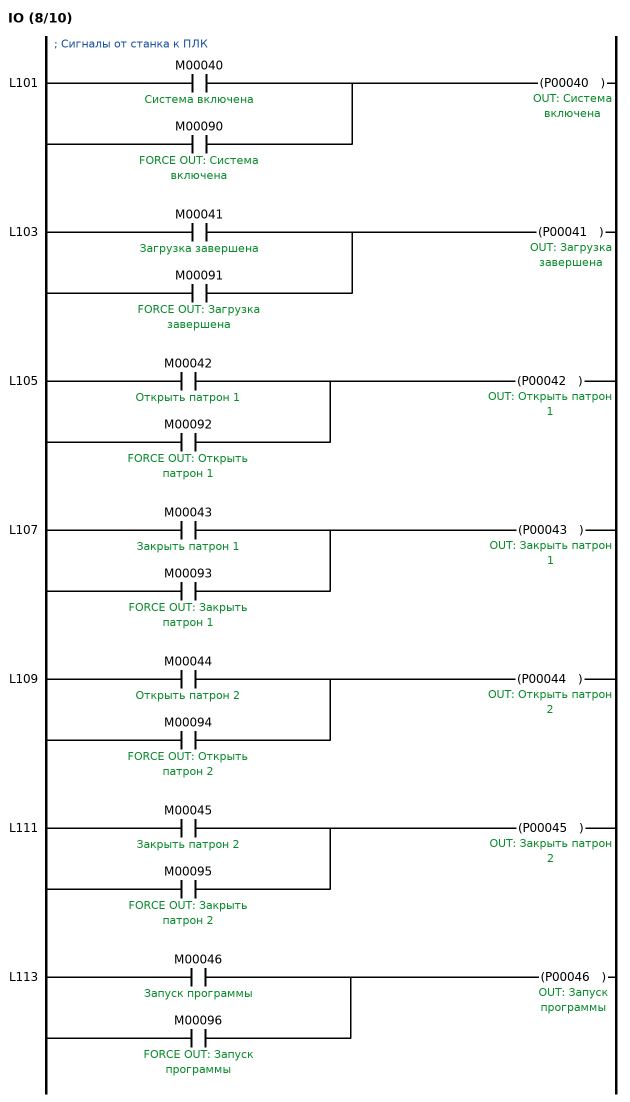
// Сигналы от станка к ПЛК
; L101
LOAD      M00040	// Система включена
OR        M00090	// FORCE OUT: Система включена
OUT       P00040	// OUT: Система включена
; L103
LOAD      M00041	// Загрузка завершена
OR        M00091	// FORCE OUT: Загрузка завершена
OUT       P00041	// OUT: Загрузка завершена
; L105
LOAD      M00042	// Открыть патрон 1
OR        M00092	// FORCE OUT: Открыть патрон 1
OUT       P00042	// OUT: Открыть патрон 1
; L107
LOAD      M00043	// Закрыть патрон 1
OR        M00093	// FORCE OUT: Закрыть патрон 1
OUT       P00043	// OUT: Закрыть патрон 1
; L109
LOAD      M00044	// Открыть патрон 2
OR        M00094	// FORCE OUT: Открыть патрон 2
OUT       P00044	// OUT: Открыть патрон 2
; L111
LOAD      M00045	// Закрыть патрон 2
OR        M00095	// FORCE OUT: Закрыть патрон 2
OUT       P00045	// OUT: Закрыть патрон 2
; L113
LOAD      M00046	// Запуск программы
OR        M00096	// FORCE OUT: Запуск программы
OUT       P00046	// OUT: Запуск программы

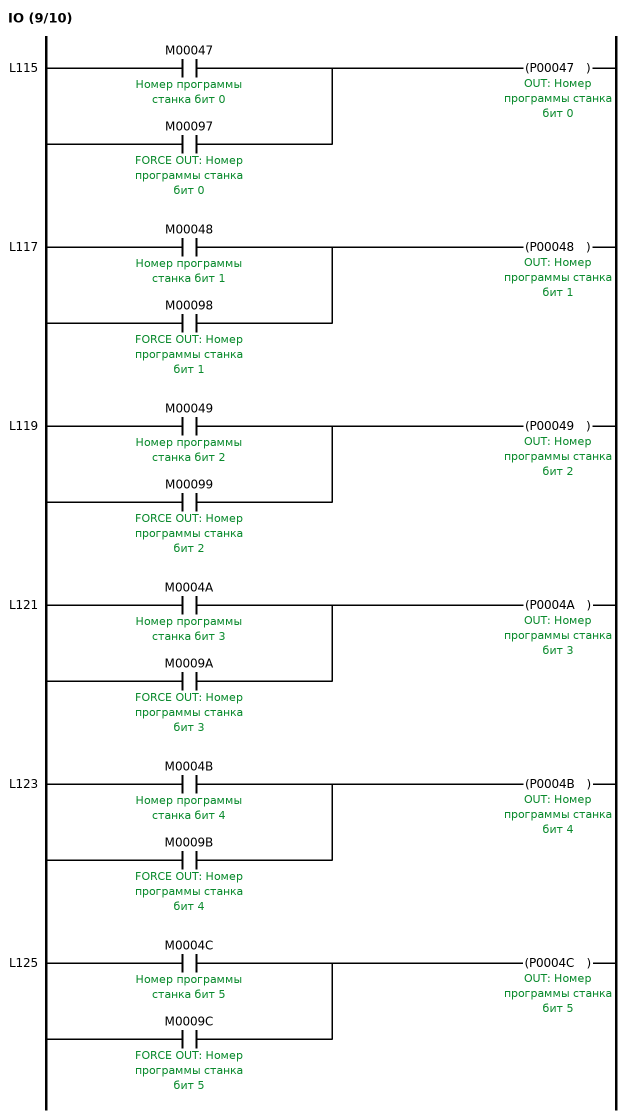
; L115
LOAD      M00047	// Номер программы станка бит 0
OR        M00097	// FORCE OUT: Номер программы станка бит 0
OUT       P00047	// OUT: Номер программы станка бит 0
; L117
LOAD      M00048	// Номер программы станка бит 1
OR        M00098	// FORCE OUT: Номер программы станка бит 1
OUT       P00048	// OUT: Номер программы станка бит 1
; L119
LOAD      M00049	// Номер программы станка бит 2
OR        M00099	// FORCE OUT: Номер программы станка бит 2
OUT       P00049	// OUT: Номер программы станка бит 2
; L121
LOAD      M0004A	// Номер программы станка бит 3
OR        M0009A	// FORCE OUT: Номер программы станка бит 3
OUT       P0004A	// OUT: Номер программы станка бит 3
; L123
LOAD      M0004B	// Номер программы станка бит 4
OR        M0009B	// FORCE OUT: Номер программы станка бит 4
OUT       P0004B	// OUT: Номер программы станка бит 4
; L125
LOAD      M0004C	// Номер программы станка бит 5
OR        M0009C	// FORCE OUT: Номер программы станка бит 5
OUT       P0004C	// OUT: Номер программы станка бит 5

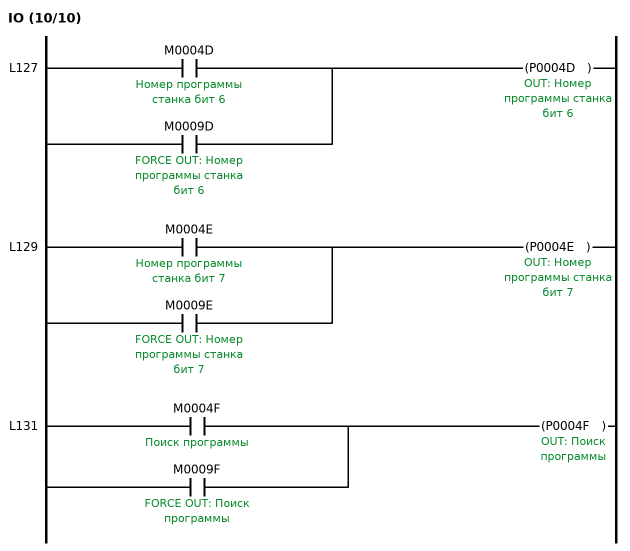
; L127
LOAD      M0004D	// Номер программы станка бит 6
OR        M0009D	// FORCE OUT: Номер программы станка бит 6
OUT       P0004D	// OUT: Номер программы станка бит 6
; L129
LOAD      M0004E	// Номер программы станка бит 7
OR        M0009E	// FORCE OUT: Номер программы станка бит 7
OUT       P0004E	// OUT: Номер программы станка бит 7
; L131
LOAD      M0004F	// Поиск программы
OR        M0009F	// FORCE OUT: Поиск программы
OUT       P0004F	// OUT: Поиск программы

PROGRAM Error (task: Scan Program)

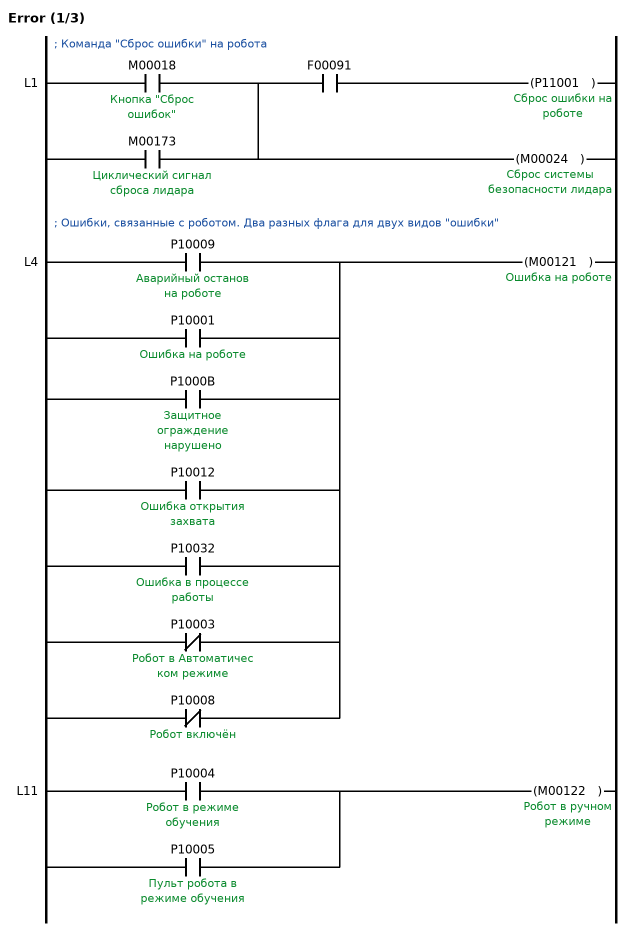
// Команда "Сброс ошибки" на робота
; L1
LOAD      M00018	// Кнопка "Сброс ошибок"
OR        M00173	// Циклический сигнал сброса лидара
MPUSH
AND       F00091
OUT       P11001	// Сброс ошибки на роботе
MPOP
OUT       M00024	// Сброс системы безопасности лидара
// Ошибки, связанные с роботом. Два разных флага для двух видов "ошибки"
; L4
LOAD      P10009	// Аварийный останов на роботе
OR        P10001	// Ошибка на роботе
OR        P1000B	// Защитное ограждение нарушено
OR        P10012	// Ошибка открытия захвата
OR        P10032	// Ошибка в процессе работы
OR NOT    P10003	// Робот в Автоматическом режиме
OR NOT    P10008	// Робот включён
OUT       M00121	// Ошибка на роботе
; L11
LOAD      P10004	// Робот в режиме обучения
OR        P10005	// Пульт робота в режиме обучения
OUT       M00122	// Робот в ручном режиме

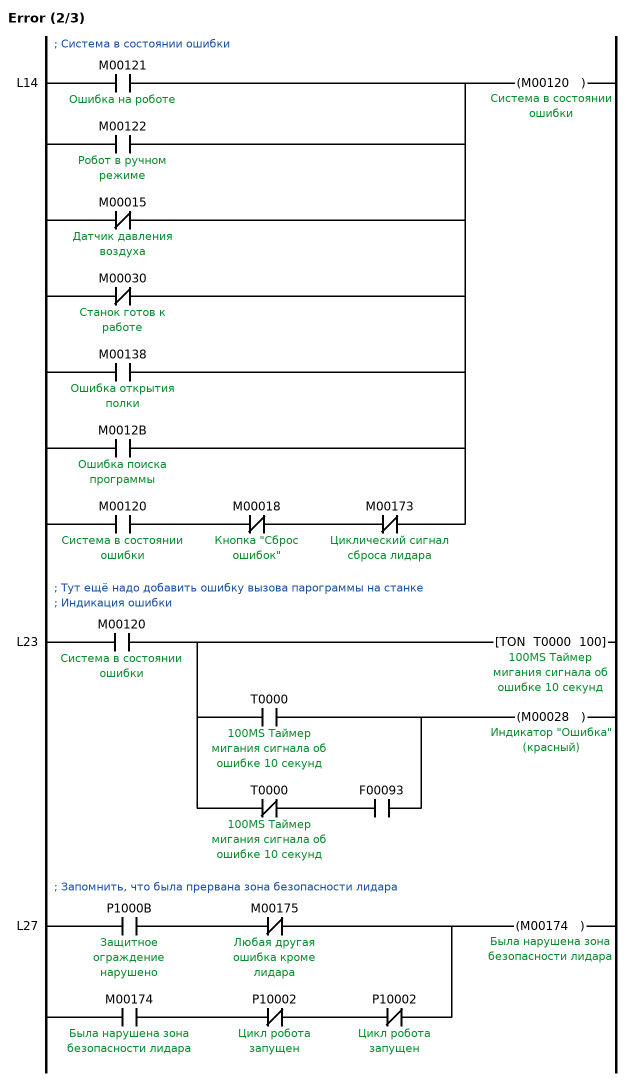
// Система в состоянии ошибки
; L14
LOAD      M00121	// Ошибка на роботе
OR        M00122	// Робот в ручном режиме
OR NOT    M00015	// Датчик давления воздуха
OR NOT    M00030	// Станок готов к работе
OR        M00138	// Ошибка открытия полки
OR        M0012B	// Ошибка поиска программы
LOAD      M00120	// Система в состоянии ошибки
AND NOT   M00018	// Кнопка "Сброс ошибок"
AND NOT   M00173	// Циклический сигнал сброса лидара
OR LOAD
OUT       M00120	// Система в состоянии ошибки
// Тут ещё надо добавить ошибку вызова парограммы на станке
// Индикация ошибки
; L23
LOAD      M00120	// Система в состоянии ошибки
TON       T0000 100	// 100MS Таймер мигания сигнала об ошибке 10 секунд
LOAD      T0000	// 100MS Таймер мигания сигнала об ошибке 10 секунд
LOAD NOT  T0000	// 100MS Таймер мигания сигнала об ошибке 10 секунд
AND       F00093
OR LOAD
AND LOAD
OUT       M00028	// Индикатор "Ошибка" (красный)
// Запомнить, что была прервана зона безопасности лидара
; L27
LOAD      P1000B	// Защитное ограждение нарушено
AND NOT   M00175	// Любая другая ошибка кроме лидара
LOAD      M00174	// Была нарушена зона безопасности лидара
AND NOT   P10002	// Цикл робота запущен
AND NOT   P10002	// Цикл робота запущен
OR LOAD
OUT       M00174	// Была нарушена зона безопасности лидара

